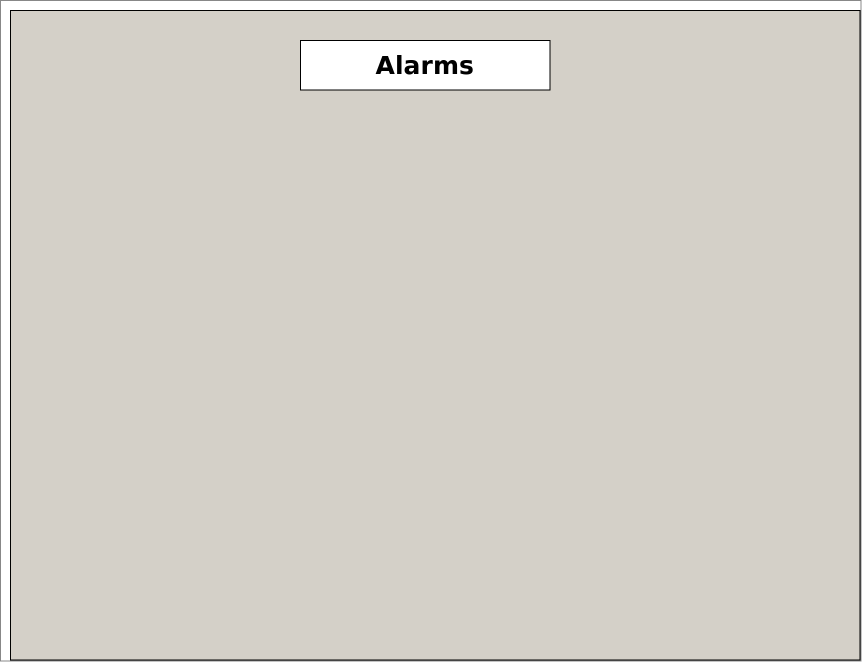
VISUALIZATION Alarms  // 862x662
    RoundedRectangle (10,10 850x650)
    RoundedRectangle (300,40 250x50), "Alarms"
END_VISUALIZATION

(* stored: Version 1.1.0.1, ProductVersion 3.1.4024.0
   Visu Alarms: Id {6dbf649e-f0ee-4e9e-8a7c-95c517abd098} *)
